TYPE ST_Euchner_MBM_HW_OUT :
STRUCT
	///Hardware Out
	nByte0: USINT;
END_STRUCT
END_TYPE

(* stored: Version 1.1.0.1, ProductVersion 3.1.4024.12
   DUT ST_Euchner_MBM_HW_OUT: Id {53cdce1a-e086-4cd6-a162-db0cbabaf464} *)
